               //step code                                             //do step
               ;
               IF #ContEnable = true THEN                               //enable continue function
                   #cont_enable[1] := true;
               END_IF;
               IF #EndOfStep = true THEN                                //define end of step condition
                   #end_of_step[1] := true;                            
               END_IF;                                    
               #next_step[1] := 0;                                      //define next step #
               IF #end_of_step[1] = true THEN                           //do on transition
                   //transition code
                   ;
               END_IF;

   //-step-100---level--1----------------------------------------------name-(remarks)----------------------                                                 
           100 :                                                     
               IF #next_step[1] = #active_step[1] THEN                   //init step     
                   //init code 
                   ;                                                  
               END_IF;

               //step code                                             //do step
               ;
               IF #ContEnable = true THEN                               //enable continue function
                   #cont_enable[1] := true;
               END_IF;
               IF #EndOfStep = true THEN                                //define end of step condition
                   #end_of_step[1] := true;                            
               END_IF;                                    
               #next_step[1] := 0;                                      //define next step #
               IF #end_of_step[1] = true THEN                           //do on transition
                   //transition code
                   ;
               END_IF;

   //-step-200---level--1----------------------------------------------name-(remarks)----------------------                                                 
           200 :                                                     
               IF #next_step[1] = #active_step[1] THEN                   //init step     
                   //init code 
                   ;                                                  
               END_IF;

               //step code                                             //do step
               ;
               IF #ContEnable = true THEN                               //enable continue function
                   #cont_enable[1] := true;
               END_IF;
               IF #EndOfStep = true THEN                                //define end of step condition
                   #end_of_step[1] := true;                            
               END_IF;                                    
               #next_step[1] := 0;                                      //define next step #
               IF #end_of_step[1] = true THEN                           //do on transition
                   //transition code
                   ;
               END_IF;

   //-error------level--1---------------------------------------------------(error in level 1)-------------
       ELSE:                                                        
           //error code                                                //do error code
           ;        
   //------------------------------------------------------------------------------------------------------
       END_CASE;

       CASE #active_step[2] OF    //sequence level_2
   //step--0-----level--2-------------------------------------------------off--(sequence off)--------------
           0    :                                                  
                #next_step[2] := 0;

   //step--1-----level--2-------------------------------------------------hold-(test sequence)-------------
           1   :                                                       
               IF #next_step[2] = #active_step[2] THEN                   //init step     
                   //init code
                   ; 
               END_IF;

               //step code                                             //do step
               ;

   //-step-10----level--2----------------------------------------------main-(start sequence)---------------                                                 
           10  :                                                     
               IF #next_step[2] = #active_step[2] THEN                   //init step     
                   //init code 
                   ;                                                  
               END_IF;

               //step code                                             //do step
               ;
               IF #ContEnable = true THEN                               //enable continue function
                   #cont_enable[2] := true;
               END_IF;
               IF #EndOfStep = true THEN                                //define end of step condition
                   #end_of_step[2] := true;                            
               END_IF;                                    
               #next_step[1] := 0;                                      //define next step #
               IF #end_of_step[2] = true THEN                           //do on transition
                   //transition code
                   ;
               END_IF;

   //-step-100---level--2----------------------------------------------name-(remarks)----------------------                                                 
           100 :                                                     
               IF #next_step[2] = #active_step[2] THEN                   //init step     
                   //init code 
                   ;                                                  
               END_IF;

               //step code                                             //do step
               ;
               IF #ContEnable = true THEN                               //enable continue function
                   #cont_enable[2] := true;
               END_IF;
               IF #EndOfStep = true THEN                                //define end of step condition
                   #end_of_step[2] := true;                            
               END_IF;                                    
               #next_step[2] := 0;                                      //define next step #
               IF #end_of_step[2] = true THEN                           //do on transition
                   //transition code
                   ;
               END_IF;

   //-error------level--2---------------------------------------------------(error in level 2)-------------
       ELSE:                                                        
           //error code                                                //do error code
           ;        
   //------------------------------------------------------------------------------------------------------
       END_CASE;

       //save crystal position at start of body - used in FB AM_RE
       //---------------------------------------------------------
       "AV".XT_POS_AT_START_BY   :=  #xt_pos_at_start;

       #start_previous := #start;                                    //save start input for next call 
       #cont_previous := "APC".CONT;                                  //save cont input for next call 
       #resume_previous := "APC".RESUME;                              //save resume input for next call
       #jump_previous := "APC".JUMP;                                  //save jump input for next call
       #single_previous := "APC".SINGLE;                              //save single input for next call
END_FUNCTION_BLOCK

FUNCTION_BLOCK "AM_EC"   // FB202, SCL
{ S7_Optimized_Access := 'FALSE' }
VERSION : 0.0
// --------------------------------------------------------------------------------
//     program     :    AM_EC
//     description :    apc endcone module  
//     name        :    D. Bruess
//     date        :    01.12.99
//     
//     revision    :    change default rotation direction: xtal= ccw and cruc= cw
//     name        :    G. Eibelsh鋟ser
//     date        :    26.04.00
// 
//     revision    :    
//     name        :    
//     date        :    
//                     (c)CGS
//     --------------------------------------------------------------------------------
   VAR_INPUT
      start : Bool;   // start sequence, activate step 10 (impulse triggered)
   END_VAR
   VAR
      start_previous : Bool;   // start input value of last call
      cont_previous : Bool;   // cont input value of last call
      resume_previous : Bool;   // resume input value of last call
      jump_previous : Bool;   // jump input value of last call
      single_previous : Bool;   // single input value of last call
      active_step : Array[0..7] of Int;   // active step number for sequence level 0..7
      next_step : Array[0..7] of Int;   // next step number for sequence level 0..7
      hold_step : Array[0..7] of Int;   // step number of step on hold
      end_of_step : Array[0..7] of Bool;   // active step is done flag for sequence 0..7
      EndOfStep : Bool;   // default value for active step is done flag
      cont_enable : Array[0..7] of Bool;   // enable continue function
      ContEnable : Bool;   // default value for enable continue function
      xt_pos_at_start : Real;   // crystal position at start of neck
      old_inc_xt_spd : Real;   // old increment value
      old_inc_cr_spd : Real;   // old increment value
      old_inc_xt_rot : Real;   // old increment value
      old_inc_cr_rot : Real;   // old increment value
   END_VAR
BEGIN


       "APC".STATUS := "APC".ENDCONE;                                  // set apc status               

       "AM_SEQUENCE_CTL" (start_p            := #start,               // control sequence
                        start_previous_p   := #start_previous,
                        cont_previous_p    := #cont_previous, 
                        resume_previous_p  := #resume_previous,
                        jump_previous_p    := #jump_previous,
                        single_previous_p  := #single_previous,
                        active_step_p      := #active_step, 
                        next_step_p        := #next_step,
                        hold_step_p        := #hold_step, 
                        end_of_step_p      := #end_of_step, 
                        cont_enable_p      := #cont_enable); 

       //Set the "Oxidation valve" in all Phases
       "DC".V21_OP:= DINT_TO_BOOL(REAL_TO_DINT("PAR_MAIN".EC_V21_OPEN));

       CASE #active_step[0] OF    //sequence level_0
   //step--0-----level--0-------------------------------------------------off--(sequence off)--------------
           0    :                                                  
                #next_step[0] := 0;

   //step--1-----level--0-------------------------------------------------hold-(test sequence)-------------
           1   :                                                       
               IF #next_step[0] = #active_step[0] THEN                   //init step     
                   //init code
                   ; 
               END_IF;

               //step code                                             //do step
               ;

   //-step-10----level--0----------------------------------------------main-(start sequence)---------------                                                 

   //-step-10----level--0-------------------------------------------------------------                                                 
   //            EC: init endcone sequence
   //---------------------------------------------------------------------------------                                                 
           10  :                                                  
               // save data of grown body (for 2nd body)
               // --------------------------------------
               IF ("APC".PNBDY = TRUE) THEN
                   "APC".LEN2_CALC := FALSE;
                   "CM_SAVE_GROWN_BY" (with_endcone := TRUE,
                                     dia          := "AC".SET_XT_DIA,
                                     len          := "AV".ACT_XT_LEN);
               END_IF;

               // init vacuum system
               // ------------------
               "DC".V1_OP    := TRUE;                         // open V1
               "DC".V3_OP    := FALSE;
               "DC".V4_OP    := FALSE;
               "DC".V5_OP    := TRUE;                         // open V5
               "DC".V6_OP    := FALSE;
               "DC".V8_OP    := FALSE;
               "DC".V11_OP   := FALSE;
               "DC".V11_CL   := TRUE;
               "DC".V12_OP   := FALSE;
               "DC".V13_OP   := FALSE;
               "DC".V20_OP   := FALSE;
               "DC".V22_OP   := FALSE;
               "DC".V24_OP   := FALSE;
               "DC".P1_ON    := TRUE;                         // start main pump
               "DC".P3_ON    := FALSE;
               "DC".V3_4_OP  := FALSE;
               "DC".V1_1_REL := FALSE;

               "DC".V1_OPEN_REQ   := FALSE;                // only EKZ 2700
               "DC".V1_CLOSE_REQ  := FALSE;

               "DC".V3_2_OP := FALSE;                      // vacuum valve feeder

               // init drives
               // -----------
               IF (("CNF".ACT_DVC_CNF AND 2#0100_0000_0000_0000_0000_0000_0000_0000) = 2#0100_0000_0000_0000_0000_0000_0000_0000) THEN   //gap control activated
                   ;                                   //direction is set in step 250 (related to gap control)
               ELSE
                   "DC".XT_LFT_UP := TRUE;               // crystal lift up - direction is set in step 250 (related to gap control)
                   "DC".XT_LFT_DN := FALSE;
                   "DC".CR_LFT_UP := TRUE;               // crucible lift up - direction is set in step 250 (related to gap control)
                   "DC".CR_LFT_DN := FALSE;
               END_IF;

               "DC".XT_LFT_FST := FALSE;
               "DC".XT_ROT_CW := "BM_ROT_DRV_DIR_DB".ROT_DIR;            //1 = cw
               "DC".XT_ROT_CCW := NOT "BM_ROT_DRV_DIR_DB".ROT_DIR;       //0 = ccw

               "DC".CR_LFT_FST := FALSE;
               "DC".CR_ROT_CW := NOT "BM_ROT_DRV_DIR_DB".ROT_DIR;        //0 = cw
               "DC".CR_ROT_CCW := "BM_ROT_DRV_DIR_DB".ROT_DIR;           //1 = ccw


               "AC".SET_XT_SPD := "CTL".SET_XT_SPD;                
               "AC".SET_XT_ROT := "KYA".SET_XT_ROT;
               "AC".SET_CR_SPD := "CTL".SET_CR_SPD;
               "AC".SET_CR_ROT := "KYA".SET_CR_ROT;

               // init heater
               // -----------
               "DC".HTR_1_ON := TRUE;                     // heater on
               "DC".HTR_2_ON := TRUE;
               "DC".HTR_3_ON := FALSE;

               // AC.SET_HTR_1_PWR := 0.0;                 do not set, loop is on
               // AC.SET_HTR_2_PWR := 0.0;
               // AC.SET_HTR_3_PWR := 0.0;

               //mobile feeder
               //-------------
               "DC".MOB_FDR_MVE_IN_SEQ_ON    :=  FALSE;
               IF ("LT".MOB_FDR_DCK_DONE AND ("DV".FDG_MVE_IN_SEQ_DONE OR NOT "DV".FDG_MVE_OUT_SEQ_DONE)) THEN 
                   "DC".MOB_FDR_MVE_OUT_SEQ_ON   :=  TRUE;
               ELSE
                   "DC".MOB_FDR_MVE_OUT_SEQ_ON   :=  FALSE;
               END_IF;
               "DC".MOB_FDR_VIB_ON           :=  FALSE;
               "FLT".MOB_FDR_NOT_DCK         :=  FALSE;
               "FLT".MOB_FDR_STP_PARA        :=  FALSE;

               // init magnet
               // -----------
               "DC".MAG_ON := ("AC".SET_MAG_1_CUR > 0.0);

               "AC".SET_MAG_1_CUR := "KYA".SET_MAG_1_CUR;
               "AC".SET_MAG_2_CUR := "KYA".SET_MAG_1_CUR * "KYA".SET_MAG_RATIO_CUR;

               // init control loops
               // ------------------
               "DC".CTL_DIA_ON       := FALSE;             // all control loops off
               "DC".CTL_GRW_RTE_ON   := FALSE;
               "DC".CTL_PULL_RTE_ON  := FALSE;
               "DC".CTL_CRUC_ROT_ON  := FALSE;
               "DC".CTL_MLT_LVL_ON   := FALSE;
               "DC".CTL_MLT_1_TMP_ON := FALSE;
               "DC".CTL_MLT_2_TMP_ON := FALSE;
               "DC".CTL_MLT_DRIFT_ON := FALSE;
               "DC".CTL_GAP_ON       := FALSE;

               "DC".CTL_HTR_1_TMP_ON := TRUE;              // heater temp loop on
               //  DC.CTL_HTR_2_TMP_ON := TRUE;

               "DC".SET_HTR_1_TMP_ABS := FALSE;                // enable inc functions
               "DC".SET_HTR_2_PWR_ABS := FALSE;


               "DC".CTL_PRS_ON := TRUE;                    // pressure control on

               "DC".CTL_SI_FDR_ON := FALSE;
               "DC".CTL_DOP_FDR_ON := FALSE;

               "DV".TRANS_SH_BY_FLAG := FALSE;
               "DV".START_SH_FLAG    := FALSE;

               "AC".SET_XT_DIA := 0.0;
               "AC".SET_GRW_RTE := 0.0;
               "AC".SET_AVG_SPD := 0.0;
               "AC".SET_AVG_CRUC_ROT := 0.0;
               "AC".SET_MLT_LVL_LSR := 0.0;
               "AC".SET_MLT_1_TMP := 0.0;
               "AC".SET_MLT_2_TMP := 0.0;

               // init measurement system
               // -----------------------
               "DC".CAM_ISP_ON   :=  TRUE;      //inspection on
               "DC".CAM_INIT     :=  FALSE;
               "DC".CAM_MLT      :=  TRUE;
               "DC".CAM_DIP      :=  FALSE;
               "DC".CAM_DIA      :=  FALSE;
               "DC".CAM_SEL_1    :=  TRUE;
               "DC".CAM_SEL_2    :=  FALSE;

               //set measurement window in upper left corner of image - no measurement required
               //------------------------------------------------------------------------------
               "AC".SET_SEN_THR    := 50.0;  
               "AC".SET_SEN_WDH    :=  5.0;        
               "AC".SET_SEN_HGT    :=  5.0;       
               "AC".SET_SEN_CTR_X  := 10.0;       
               "AC".SET_SEN_CTR_Y  := 10.0;  

               "DV".THR_CALC_DISABLED  := TRUE;      //threshold calculation in this step is disabled

               "DC".LSR_ON := FALSE;                       // laser off
               "DC".MCC_ON := FALSE;                       // melt contact control off
               "DC".MCC_TST_ON := FALSE;

               // init Si feeder system
               // ---------------------
               "DC".SI_FDR_ON := FALSE;                    // feeder off
               "DC".DOP_FDR_ON := FALSE;

               "AC".SET_FDR_SI := 0.0;
               "AC".SET_FDR_DOP := 0.0;

               // init lamp on control cabinet
               // ----------------------------
               "DV".LMP_OR := false;

               // save start position, reset length
               // ---------------------------------
               #xt_pos_at_start := "AV".ACT_XT_POS;
               "AV".ACT_XT_LEN_PRC := 0.0; 
               "AV".ACT_XT_LEN := 0.0;

               // calculate all setpoints 
               // -----------------------
               "AM_PAR_FNC_EC" (act_x_value := 0);



               // enable automatic mode
               // ---------------------
               "DC".MOD_AUT_ENB := TRUE;

               #end_of_step[0]  := true;                            
               #next_step[0]    := 100;

   //-step-100---level--0-------------------------------------------------------------                                                 
   //            EC: wait for automatic mode
   //---------------------------------------------------------------------------------                                                 
           100 :                                                     
               IF #next_step[0] = #active_step[0] THEN
                   "APC".OP_MSG := "OP_MSG".WAIT_FOR_AUTO;                                                  
               END_IF;

               // do not count the length while waiting for automatic
               // ---------------------------------------------------
               #xt_pos_at_start := "AV".ACT_XT_POS;
               "AV".ACT_XT_LEN_PRC := 0.0; 
               "AV".ACT_XT_LEN := 0.0;

               // calculate all setpoints 
               // -----------------------
               "AM_PAR_FNC_EC" (act_x_value := 0.0);

               IF "APC".AUTOMATIC = TRUE THEN                     // automatic mode ?
                   #end_of_step[0] := true;                            
               END_IF;                                    
               #next_step[0] := 200;

   //-step-200---level--0-------------------------------------------------------------                                                 
   //            EC: start time
   //---------------------------------------------------------------------------------                                                 
           200 :                                                     
               "APC".ACT_TME_PROC := 0;                           // start process time
               "APC".ACT_TME_STE := 0;                            // reset time of step
               "APC".TI[0] := 0;                                  // start waiting time
               "APC".OP_MSG := "OP_MSG".BLANK;                                                  

               #end_of_step[0] := true;

               IF (("CNF".ACT_DVC_CNF AND 2#0100_0000_0000_0000_0000_0000_0000_0000) = 2#0100_0000_0000_0000_0000_0000_0000_0000) THEN   //gap control activated
                   #next_step[0] := 250;
               ELSE
                   #next_step[0] := 300;
               END_IF;

   //-step-250---level--0-------------------------------------------------------------                                                 
   //            EC: set lifting direction related to speed set points
   //---------------------------------------------------------------------------------                                                 
           250 :                                                     
               //Set direction of crystal lift
               //-----------------------------
               IF (("CTL".SET_XT_SPD + "AV".MLT_LVL_SFT_OFFS_SPD + "CTL".SET_SPEED_OFFS) < 0.0) THEN
                   "DC".XT_LFT_UP    := FALSE;
                   "DC".XT_LFT_DN    := TRUE; // crystal lift down
                   "LT".XT_LFT_UP    := FALSE;
               ELSE
                   "DC".XT_LFT_UP    := TRUE; // crystal lift up
                   "DC".XT_LFT_DN    := FALSE;
                   "LT".XT_LFT_DN    := FALSE;
               END_IF;
               //Set direction of crucible lift
               //------------------------------
               IF (("CTL".SET_CR_SPD + "AV".MLT_LVL_SFT_OFFS_SPD + "CTL".SET_SPEED_OFFS ) < 0.0) THEN
                   "DC".CR_LFT_UP    := FALSE;
                   "DC".CR_LFT_DN    := TRUE; // Crucible lift down
                   "LT".CR_LFT_UP    := FALSE;
               ELSE
                   "DC".CR_LFT_UP    := TRUE; // Crucible lift up
                   "DC".CR_LFT_DN    := FALSE;
                   "LT".CR_LFT_DN    := FALSE;
               END_IF;

               //lifitng direction upwads active?
               // -------------------------------
               IF ("DC".XT_LFT_UP AND "DC".CR_LFT_UP) THEN    
                   #end_of_step[0] := true;                            
               END_IF;

               #next_step[0] := 300; 

   //-step-300---level--0-------------------------------------------------------------                                                 
   //            EC: do initial inc. for speed, rotation and heater
   //---------------------------------------------------------------------------------                                                 
           300 :                                                     
               IF #next_step[0] = #active_step[0] THEN                       
                   //display initial temperature and power setpoints
                   //-----------------------------------------------
                   "DIS".HTR_1_TMP_SET_PHA_STR   :=  "CTL".SET_HTR_1_TMP;
                   "DIS".HTR_2_PWR_SET_PHA_STR   :=  "CTL".SET_HTR_2_PWR;
                   // do heater inc.
                   // --------------
                   "DC".RSTRT_HTR_1_TMP_INC := TRUE;
                   "DC".RSTRT_HTR_2_PWR_INC := TRUE;
                   "AC".SET_HTR_1_TMP_INC := "AV".SET_HTR_1_TMP_INC;
                   "AC".SET_HTR_2_PWR_INC := "AV".SET_HTR_2_PWR_INC;
               END_IF;

               // calculate actual length
               // -----------------------
               "AM_CALC_LENGTH" (start_pos := #xt_pos_at_start,
                               actual_pos := "AV".ACT_XT_POS,
                               total_len := "PAR_MAIN".EC_XT_LEN,
                               actual_len => "AV".ACT_XT_LEN,
                               actual_len_prc => "AV".ACT_XT_LEN_PRC);


               // calculate all setpoints for this step
               // -------------------------------------                                      
               "AM_PAR_FNC_EC" (act_x_value := "AV".ACT_XT_LEN);

               // setpoint magnet
               // ---------------
               "DC".MAG_ON := ("AC".SET_MAG_1_CUR > 0.0);

               "AC".SET_MAG_1_CUR := "AV".SET_MAG_1_CUR;
               "AC".SET_MAG_2_CUR := "AV".SET_MAG_1_CUR * "AV".SET_MAG_RATIO_CUR;



               // reset waiting time 1 for oxidation process
               //-------------------------------------------
               "APC".TI[1] := 0;

               // wait ?
               // ------
               IF ("APC".TI[0] > 3) THEN    
                   #end_of_step[0] := true;                            
               END_IF;
               #next_step[0] := 400; 


   //-step-400---level--0-------------------------------------------------------------                                                 
   //            EC: do endcone process
   //---------------------------------------------------------------------------------                                                 
           400 :                                                  
               IF #next_step[0] = #active_step[0] THEN                       
                   // init inc. functions
                   // -------------------
                   #old_inc_xt_spd := 0.0;
                   #old_inc_cr_spd := 0.0;
                   #old_inc_xt_rot := 0.0;
                   #old_inc_cr_rot := 0.0;
               END_IF;

               // calculate actual length
               // -----------------------
               "AM_CALC_LENGTH" (start_pos      := #xt_pos_at_start,
                               actual_pos     := "AV".ACT_XT_POS,
                               total_len      := "PAR_MAIN".EC_XT_LEN,
                               actual_len     => "AV".ACT_XT_LEN,
                               actual_len_prc => "AV".ACT_XT_LEN_PRC);

               // calculate all setpoints for this step
               // -------------------------------------                                      
               "AM_PAR_FNC_EC" (act_x_value := "AV".ACT_XT_LEN);

               // setpoint magnet
               // ---------------
               "DC".MAG_ON := ("AC".SET_MAG_1_CUR > 0.0);

               "AC".SET_MAG_1_CUR := "AV".SET_MAG_1_CUR;
               "AC".SET_MAG_2_CUR := "AV".SET_MAG_1_CUR * "AV".SET_MAG_RATIO_CUR;

               // increment function for speed and rotation
               // -----------------------------------------
               "AM_CALC_INC" (inc_disable := FALSE,
                            semi        := "SY".CTL_DIA_SMI,     // semi mode for crystal lift
                            inc_new     := "AV".SET_XT_SPD,
                            setp_man    := "KYA".SET_XT_SPD,
                            setp_min    := 0.0,                
                            setp_max    := "CNF".XT_LFT_RANGE,
                            setp_out    := "AC".SET_XT_SPD,
                            inc_old     := #old_inc_xt_spd );

               "AM_CALC_INC" (inc_disable := FALSE,
                            semi        := "SY".CTL_CR_SPD_SMI,
                            inc_new     := "AV".SET_CR_SPD,
                            setp_man    := "KYA".SET_CR_SPD,
                            setp_min    := 0.0,
                            setp_max    := "CNF".CR_LFT_RANGE,
                            setp_out    := "AC".SET_CR_SPD,
                            inc_old     := #old_inc_cr_spd );

               "AM_CALC_INC" (inc_disable := ("PAR_MAIN".EC_ROT_ABS_INC = 1.0), 
                            semi        := "SY".CTL_XT_ROT_SMI,  
                            inc_new     := "AV".SET_XT_ROT,
                            setp_man    := "KYA".SET_XT_ROT,
                            setp_min    := 0.0,
                            setp_max    := "CNF".XT_ROT_RANGE,
                            setp_out    := "AC".SET_XT_ROT,
                            inc_old     := #old_inc_xt_rot );

               "AM_CALC_INC" (inc_disable := ("PAR_MAIN".EC_ROT_ABS_INC = 1.0),
                            semi        := "SY".CTL_CR_ROT_SMI,  
                            inc_new     := "AV".SET_CR_ROT,
                            setp_man    := "KYA".SET_CR_ROT,
                            setp_min    := 0.0,
                            setp_max    := "CNF".CR_ROT_RANGE,
                            setp_out    := "AC".SET_CR_ROT,
                            inc_old     := #old_inc_cr_rot );

               // heater temp/power inc.
               // ----------------------
               "AC".SET_HTR_1_TMP_INC := "AV".SET_HTR_1_TMP_INC;
               "AC".SET_HTR_2_PWR_INC := "AV".SET_HTR_2_PWR_INC;

               // melt contact control
               // --------------------   
               "DC".MCC_ON := ("PAR_MAIN".EC_MLT_CONTACT_CTL = 1.0);     

               // endcone length reached ?
               // ------------------------
               IF ("AV".ACT_XT_LEN >= "PAR_MAIN".EC_XT_LEN) THEN    
                   #end_of_step[0] := true;                            
               END_IF;
               #next_step[0] := 500;


   //-step-500---level--0-------------------------------------------------------------                                                 
   //            EC: start shut down process
   //---------------------------------------------------------------------------------                                                 
           500 :                                                  
               IF #next_step[0] = #active_step[0] THEN
                   "APC".OP_MSG := "OP_MSG".BLANK;
               END_IF;

               IF ("APC".SUTDN = TRUE) THEN
                   "DC".MOD_SD := TRUE;                           // switch to shut down 
               ELSE
                   "DC".MOD_RE := TRUE;                           // switch to removal 
               END_IF;   
               #next_step[0] := 500;                             // E N D 



   //---------------------------------------------------------------------------------                                                 
   //-error------level--0---------------------------------------------------(error in level 0)-------------
       ELSE:                                                        
           //error code                                                //do error code
           ;        
   //------------------------------------------------------------------------------------------------------
       END_CASE;

       #start_previous := #start;                                    //save start input for next call 
       #cont_previous := "APC".CONT;                                  //save cont input for next call 
       #resume_previous := "APC".RESUME;                              //save resume input for next call
       #jump_previous := "APC".JUMP;                                  //save jump input for next call
       #single_previous := "APC".SINGLE;                              //save single input for next call
END_FUNCTION_BLOCK

FUNCTION_BLOCK "AM_SD"   // FB203, SCL
{ S7_Optimized_Access := 'FALSE' }
VERSION : 0.0
// --------------------------------------------------------------------------------
//     program     :    AM_SD
//     description :    apc shut down module  
//     name        :    D. Bruess
//     date        :    18.11.99
//     
//     revision    :    change default rotation direction: xtal= ccw and cruc= cw
//     name        :    G. Eibelsh鋟ser
//     date        :    26.04.00
// 
//     revision    :    
//     name        :    
//     date        :    
//                     (c)PVA TePla AG
//     --------------------------------------------------------------------------------
   VAR_INPUT
      start : Bool;   // start sequence, activate step 10 (impulse triggered)
   END_VAR
   VAR
      start_previous : Bool;   // start input value of last call
      cont_previous : Bool;   // cont input value of last call
      resume_previous : Bool;   // resume input value of last call
      jump_previous : Bool;   // jump input value of last call
      single_previous : Bool;   // single input value of last call
      active_step : Array[0..7] of Int;   // active step number for sequence level 0..7
      next_step : Array[0..7] of Int;   // next step number for sequence level 0..7
      hold_step : Array[0..7] of Int;   // step number of step on hold
      end_of_step : Array[0..7] of Bool;   // active step is done flag for sequence 0..7
      EndOfStep : Bool;   // default value for active step is done flag
      cont_enable : Array[0..7] of Bool;   // enable continue function
      ContEnable : Bool;   // default value for enable continue function
      cruc_in_pos : Bool;   // crucible in new position
      xtal_in_pos : Bool;   // crystal in new position
      prs_ctl_done : Bool;   // new pressure reached
      v4_lim_reached : Bool;   // pressure limit for gas inlet through V4 is reached
      OV2 : Bool;   // ???????
      par_line : Int;   // act. line from parameter table
      par_step : Int;   // number of this step
      par_time : Int;   // time parameter for this step
      set_cr_pos_old : Real;   // old setpoint for crucible position
      set_xt_pos_old : Real;   // old setpoint for crystal position
      set_clf_prs_old : Real;   // old setpoint for pressure
      set_gas_1_flw_old : Real;   // old setpoint for gas flow
      set_gas_2_flw_old : Real;   // old setpoint for gas flow
      prs_leak_test_start : Real;   // pressure at start of leak test
   END_VAR
BEGIN


       "APC".STATUS := "APC".SHUT_DOWN;                                // set apc status               

       "AM_SEQUENCE_CTL" (start_p            := #start,               // control sequence
                        start_previous_p   := #start_previous,
                        cont_previous_p    := #cont_previous, 
                        resume_previous_p  := #resume_previous,
                        jump_previous_p    := #jump_previous,
                        single_previous_p  := #single_previous,
                        active_step_p      := #active_step, 
                        next_step_p        := #next_step,
                        hold_step_p        := #hold_step, 
                        end_of_step_p      := #end_of_step, 
                        cont_enable_p      := #cont_enable); 


       CASE #active_step[0] OF    //sequence level_0
   //step--0-----level--0-------------------------------------------------off--(sequence off)--------------
           0    :                                                  
                #next_step[0] := 0;

   //step--1-----level--0-------------------------------------------------hold-(test sequence)-------------
           1   :                                                       
               IF #next_step[0] = #active_step[0] THEN                   //init step     
                   //init code
                   ; 
               END_IF;

               //step code                                             //do step
               ;

   //-step-10----level--0----------------------------------------------main-(start sequence)---------------                                                 

   //-step-10----level--0-------------------------------------------------------------                                                 
   //            SD: init shut down sequence
   //---------------------------------------------------------------------------------                                                 
           10  :                                                     

               // init vacuum system
               // ------------------
               "DC".V3_OP    := FALSE;
               "DC".V3_2_OP  := FALSE;                      // vacuum valve feeder
               "DC".V4_OP    := FALSE;
               "DC".V5_OP    := TRUE;                         // open V5
               "DC".V6_OP    := FALSE;
               "DC".V8_OP    := FALSE;
               "DC".V11_OP   := FALSE;
               "DC".V11_CL   := TRUE;
               "DC".V12_OP   := FALSE;
               "DC".V13_OP   := FALSE;
               "DC".V20_OP   := FALSE;
               "DC".V21_OP   := DINT_TO_BOOL(REAL_TO_DINT("PAR_MAIN".SD_V21_OPEN));    //Set the Oxidation valve according parameter
               "DC".V22_OP   := FALSE;
               "DC".V24_OP   := FALSE;
               "DC".P1_ON    := TRUE;                         // start main pump
               "DC".P3_ON    := FALSE;
               "DC".V1_OPEN_REQ   := FALSE;                // only EKZ 2700
               "DC".V1_CLOSE_REQ  := FALSE;
               "DC".V3_4_OP  := FALSE;
               "DC".V1_1_REL := FALSE;

               #set_clf_prs_old  := -1.0; 
               #set_gas_1_flw_old:= -1.0;
               #set_gas_2_flw_old:= -1.0;
               #prs_ctl_done := FALSE;
               "AM_PRS_CTRL_DB".req_vac := FALSE;
               "AM_PRS_CTRL_DB".req_vent := FALSE;

               // init drives
               // -----------
               "DC".XT_LFT_UP  := FALSE;                    // stop crystal lift
               "DC".XT_LFT_DN  := FALSE;
               "DC".XT_LFT_FST := FALSE;
               "DC".XT_ROT_CW  := "BM_ROT_DRV_DIR_DB".ROT_DIR      AND ("AC".SET_XT_ROT <> 0.0);    //1 = cw
               "DC".XT_ROT_CCW := NOT "BM_ROT_DRV_DIR_DB".ROT_DIR  AND ("AC".SET_XT_ROT <> 0.0);    //0 = ccw


               "DC".CR_LFT_UP  := FALSE;                    // stop crucible lift
               "DC".CR_LFT_DN  := FALSE;
               "DC".CR_LFT_FST := FALSE;
               "DC".CR_ROT_CW  := NOT "BM_ROT_DRV_DIR_DB".ROT_DIR  AND ("AC".SET_CR_ROT <> 0.0);     //0 = cw
               "DC".CR_ROT_CCW := "BM_ROT_DRV_DIR_DB".ROT_DIR      AND ("AC".SET_CR_ROT <> 0.0);     //1 = ccw


               "AC".SET_XT_SPD := 0.0;                
               "AC".SET_XT_ROT := "KYA".SET_XT_ROT;
               "AC".SET_CR_SPD := 0.0;
               "AC".SET_CR_ROT := "KYA".SET_CR_ROT;

               #set_cr_pos_old := -1.0;
               #set_xt_pos_old := -1.0;
               #cruc_in_pos := FALSE;
               #xtal_in_pos := FALSE;
               "AM_CR_DRV_MOVE_DB".pos_req := FALSE;
               "AM_XT_DRV_MOVE_DB".pos_req := FALSE;

               // init heater
               // -----------
               "DC".HTR_1_ON := ("AC".SET_HTR_1_PWR > 0.0);    // heater on
               "DC".HTR_2_ON := FALSE;                       // heater off
               "DC".HTR_3_ON := FALSE;

               "AC".SET_HTR_1_PWR := "KYA".SET_HTR_1_PWR;
               "AC".SET_HTR_2_PWR := 0.0;
               "AC".SET_HTR_3_PWR := 0.0;

               //mobile feeder
               //-------------
               "DC".MOB_FDR_MVE_IN_SEQ_ON    :=  FALSE;
               IF ("LT".MOB_FDR_DCK_DONE AND ("DV".FDG_MVE_IN_SEQ_DONE OR NOT "DV".FDG_MVE_OUT_SEQ_DONE)) THEN 
                   "DC".MOB_FDR_MVE_OUT_SEQ_ON   :=  TRUE;
               ELSE
                   "DC".MOB_FDR_MVE_OUT_SEQ_ON   :=  FALSE;
               END_IF;
               "DC".MOB_FDR_VIB_ON           :=  FALSE;
               "FLT".MOB_FDR_NOT_DCK         :=  FALSE;
               "FLT".MOB_FDR_STP_PARA        :=  FALSE;

               // init magnet
               // -----------
               "DC".MAG_ON := ("AC".SET_MAG_1_CUR > 0.0);

               "AC".SET_MAG_1_CUR := "KYA".SET_MAG_1_CUR;            
               "AC".SET_MAG_2_CUR := "KYA".SET_MAG_1_CUR * "KYA".SET_MAG_RATIO_CUR;

               // init control loops
               // ------------------
               "DC".CTL_DIA_ON := FALSE;                   // all control loops off
               "DC".CTL_GRW_RTE_ON := FALSE;
               "DC".CTL_PULL_RTE_ON := FALSE;
               "DC".CTL_CRUC_ROT_ON := FALSE;
               "DC".CTL_MLT_LVL_ON := FALSE;
               "DC".CTL_MLT_1_TMP_ON := FALSE;
               "DC".CTL_MLT_2_TMP_ON := FALSE;
               "DC".CTL_MLT_DRIFT_ON := FALSE;
               "DC".CTL_GAP_ON       := FALSE;

               "DC".CTL_HTR_1_TMP_ON := FALSE;
               // DC.CTL_HTR_2_TMP_ON := FALSE;

               "DC".SET_HTR_1_TMP_ABS := TRUE;             // disable inc functions
               "DC".SET_HTR_2_PWR_ABS := TRUE;


               "DC".CTL_PRS_ON := TRUE;                    // pressure control on

               "DC".CTL_SI_FDR_ON := FALSE;
               "DC".CTL_DOP_FDR_ON := FALSE;

               "DV".TRANS_SH_BY_FLAG := FALSE;
               "DV".START_SH_FLAG    := FALSE;


               "AC".SET_XT_DIA := 0.0;
               "AC".SET_GRW_RTE := 0.0;
               "AC".SET_AVG_SPD := 0.0;
               "AC".SET_AVG_CRUC_ROT := 0.0;
               "AC".SET_MLT_LVL_LSR := 0.0;
               "AC".SET_MLT_1_TMP := 0.0;
               "AC".SET_MLT_2_TMP := 0.0;
               "AC".SET_HTR_1_TMP := 0.0;
               "AC".SET_HTR_2_TMP := 0.0;

               // init measurement system
               // -----------------------
               "DC".CAM_ISP_ON   :=  FALSE;      //inspection off
               "DC".CAM_INIT     :=  FALSE;
               //DC.CAM_MLT      :=  FALSE;
               //DC.CAM_DIP      :=  FALSE;
               //DC.CAM_DIA      :=  TRUE;
               "DC".CAM_SEL_1    :=  TRUE;
               "DC".CAM_SEL_2    :=  FALSE;

               "DV".THR_CALC_DISABLED  := TRUE;      //threshold calculation in this step is disabled


               "DC".LSR_ON := FALSE;                       // laser off
               "DC".MCC_ON := FALSE;                       // melt contact control off
               "DC".MCC_TST_ON := FALSE;

               // init Si feeder system
               // ---------------------
               "DC".SI_FDR_ON := FALSE;                    // feeder off
               "DC".DOP_FDR_ON := FALSE;

               "AC".SET_FDR_SI := 0.0;
               "AC".SET_FDR_DOP := 0.0;

               // init lamp on control cabinet
               // ----------------------------
               "DV".LMP_OR := false;

               // calculate all setpoints (step no from 1st line of seqence table)
               // ----------------------------------------------------------------
               #par_line := 1;
               #par_step := REAL_TO_INT ("PAR_X_VALUES_1".PAR["APC".SHUT_DOWN, #par_line]);            
               "AM_PAR_FNC_SD" (act_x_value := #par_step);

               // process control flags
               // ---------------------
               "APC".PNBDY := FALSE;

               IF ("STA".ACT_STATE = "APC".STATE_RUN) THEN 
                   "DV".FIL_FSH_REQ_AFTER_SD :=  TRUE;           //request automtic filter flushing after shut down
               ELSE
                   "DV".FIL_FSH_REQ_AFTER_SD :=  FALSE;
               END_IF;

               // enable automatic mode
               // ---------------------
               "DC".MOD_AUT_ENB := TRUE;

               #end_of_step[0] := true;                            
               #next_step[0] := 100;


   //-step-100---level--0-------------------------------------------------------------                                                 
   //            SD: wait for automatic mode
   //---------------------------------------------------------------------------------                                                 
           100 :                                                     
               IF #next_step[0] = #active_step[0] THEN
                   "APC".OP_MSG := "OP_MSG".WAIT_FOR_AUTO;                                                  
               END_IF;

               IF "APC".AUTOMATIC = TRUE THEN                     // automatic mode ?
                   #end_of_step[0] := true;                            
               END_IF;                                    
               #next_step[0] := 150;


   //-step-150---level--0-------------------------------------------------------------                                                 
   //            SD: start time
   //---------------------------------------------------------------------------------                                                 
           150 :                                                     
               "APC".ACT_TME_PROC := 0;                           // start process time
               "APC".TI[1] := 0;                                  // reset waiting time 1 for oxidation process
               #end_of_step[0] := true;                            
               #next_step[0] := 200;


   //-step-200---level--0-------------------------------------------------------------                                                 
   //            SD: do one shut down step
   //---------------------------------------------------------------------------------                                                 
           200 :                                                     
               IF #next_step[0] = #active_step[0] THEN                       
                   //reset initial temperature and power setpoints
                   //---------------------------------------------
                   "DIS".HTR_1_TMP_SET_PHA_STR   :=  0.0;
                   "DIS".HTR_2_PWR_SET_PHA_STR   :=  0.0;

                   "APC".TI[0] := 0;                     // start step time
               END_IF;

               // fetch actual step number and time for this step
               // -----------------------------------------------
               #par_step := REAL_TO_INT ("PAR_X_VALUES_1".PAR["APC".SHUT_DOWN, #par_line]);            
               #par_time := REAL_TO_INT ("PAR_TME".PAR["APC".SHUT_DOWN, #par_line]);

               //Oxidation valve vacuum pipes
               //----------------------------
               "DC".V21_OP:= DINT_TO_BOOL(REAL_TO_DINT("PAR_MAIN".SD_V21_OPEN));

               // show actual step number
               // -----------------------
               "APC".OP_MSG := #par_step;

               // calculate all setpoints for this step
               // -------------------------------------                                      
               "AM_PAR_FNC_SD" (act_x_value := #par_step);

               // setpoint magnet
               // ---------------
               "DC".MAG_ON := ("AC".SET_MAG_1_CUR > 0.0);

               "AC".SET_MAG_1_CUR := "AV".SET_MAG_1_CUR;
               "AC".SET_MAG_2_CUR := "AV".SET_MAG_1_CUR * "AV".SET_MAG_RATIO_CUR;

               // move crucible
               // -------------
               IF ("AV".SET_CR_POS <> #set_cr_pos_old) THEN
                 #cruc_in_pos := FALSE;
               END_IF;

               "DC".CR_LFT_FST := TRUE;

               "AM_CR_DRV_MOVE_DB" ( set_pos := "AV".SET_CR_POS,
                                               set_spd := "AV".SET_CR_SPD,
                                               act_pos := "AV".ACT_CR_POS,
                                               cnf     := "CNF".CNF_CR_POS,
                                               out_up  := "DC".CR_LFT_UP,
                                               out_dn  := "DC".CR_LFT_DN,
                                               out_spd := "AC".SET_CR_SPD,
                                               done    := #cruc_in_pos);

               IF (#cruc_in_pos) THEN
                 #set_cr_pos_old := "AV".SET_CR_POS;
               END_IF;


               // move crystal
               // ------------
               IF ("AV".SET_XT_POS <> #set_xt_pos_old) THEN
                 #xtal_in_pos := FALSE;
               END_IF;

               "DC".XT_LFT_FST := TRUE;

               "AM_XT_DRV_MOVE_DB" (set_pos := "AV".SET_XT_POS,
                                           set_spd := - "AV".SET_XT_SPD,
                                           act_pos := "AV".ACT_XT_POS,
                                           cnf     := "CNF".CNF_XT_POS,
                                           out_up  := "DC".XT_LFT_DN,    // (!)
                                           out_dn  := "DC".XT_LFT_UP,    // (!)
                                           out_spd := "AC".SET_XT_SPD,
                                           done    := #xtal_in_pos);

               IF (#xtal_in_pos) THEN
                 #set_xt_pos_old := "AV".SET_XT_POS;
               END_IF;

               // control pressure and gas flow
               // -----------------------------
               IF ("AV".SET_GAS_1_FLW <> #set_gas_1_flw_old) THEN
                 #prs_ctl_done := FALSE;
               END_IF;
               IF ("AV".SET_GAS_2_FLW <> #set_gas_2_flw_old) THEN
                 #prs_ctl_done := FALSE;
               END_IF;
               IF ("AV".SET_PRS_FCH <> #set_clf_prs_old) THEN
                 #prs_ctl_done := FALSE;
               END_IF;

               "AM_PRS_CTRL_DB" (set_prs      := "AV".SET_PRS_FCH,
                                           set_flw_1    := "AV".SET_GAS_1_FLW,
                                           set_flw_2    := "AV".SET_GAS_2_FLW,
                                           act_prs      := "AV".ACT_PRS_FCH,
                                           out_V4       := "DC".V4_OP,
                                           out_V5       := "DC".V5_OP,
                                           out_prs_ctl  := "DC".CTL_PRS_ON,
                                           out_flw_1    := "AC".SET_GAS_1_FLW,
                                           out_flw_2    := "AC".SET_GAS_2_FLW,
                                           out_prs      := "AC".SET_CLF_PRS,
                                           out_valve_pos:= "AC".SET_CTL_VALVE_POS,
                                           done         := #prs_ctl_done);

               IF (#prs_ctl_done) THEN
                 #set_gas_1_flw_old := "AV".SET_GAS_1_FLW;
                 #set_gas_2_flw_old := "AV".SET_GAS_2_FLW;
                 #set_clf_prs_old := "AV".SET_PRS_FCH;
               END_IF;

               // close pressure control valve (only EKZ 2700)
               //---------------------------------------------
               IF "DC".CTL_PRS_ON = FALSE    THEN             
                   "DC".V1_OPEN_REQ   := FALSE;                
                   "DC".V1_CLOSE_REQ  := TRUE;
               ELSE
                   "DC".V1_OPEN_REQ   := FALSE;                
                   "DC".V1_CLOSE_REQ  := FALSE;
               END_IF;    

               // control heater
               // --------------
               "DC".HTR_1_ON := ("AC".SET_HTR_1_PWR > 0.0);
               "DC".HTR_2_ON := FALSE;


               // control rotation
               // ----------------
               "DC".XT_ROT_CW  := "BM_ROT_DRV_DIR_DB".ROT_DIR      AND ("AC".SET_XT_ROT <> 0.0);    //1 = cw
               "DC".XT_ROT_CCW := NOT "BM_ROT_DRV_DIR_DB".ROT_DIR  AND ("AC".SET_XT_ROT <> 0.0);    //0 = ccw
               "DC".CR_ROT_CW  := NOT "BM_ROT_DRV_DIR_DB".ROT_DIR  AND ("AC".SET_CR_ROT <> 0.0);    //0 = cw
               "DC".CR_ROT_CCW := "BM_ROT_DRV_DIR_DB".ROT_DIR      AND ("AC".SET_CR_ROT <> 0.0);    //1 = ccw


               // time till end of this step
               // --------------------------
               "APC".ACT_TME_STE := #par_time - "APC".TI[0];

               // end of step ?
               // -------------
               IF (("APC".TI[0] > #par_time)
                    AND (#cruc_in_pos = TRUE)
                    AND (#xtal_in_pos = TRUE)
                    AND (#prs_ctl_done = TRUE))  THEN

                  #end_of_step[0] := true;
               END_IF;

               #next_step[0] := 300; 


   //-step-300---level--0-------------------------------------------------------------                                                 
   //            SD: transition to next step, check for last step
   //---------------------------------------------------------------------------------                                                 
           300 :                                                  
               IF #next_step[0] = #active_step[0] THEN                       
                   // next line in parameter table
                   // ----------------------------
                   #par_line := #par_line + 1;
               END_IF;

               // fetch step number of this new line
               // ----------------------------------
               IF (#par_line <= 21) THEN
                   #par_step := REAL_TO_INT ("PAR_X_VALUES_1".PAR["APC".SHUT_DOWN, #par_line]);            
               END_IF;


               // step number = 0 or last line ? 
               // ------------------------------
               IF ((#par_step = 0)
                   OR (#par_line > 21) ) THEN

                   // start waiting time
                   // ------------------
                   #end_of_step[0] := true;                            
                   #next_step[0] := 400; 
               ELSE
                   // continue with next shut down step
                   // ---------------------------------
                   #end_of_step[0] := true;                            
                   #next_step[0] := 200; 
               END_IF;


   //-step-400---level--0-------------------------------------------------------------                                                 
   //            SD: initialisation after sequence
   //---------------------------------------------------------------------------------                                                 
           400 :                                                  
               IF #next_step[0] = #active_step[0] THEN
                   "APC".OP_MSG := "OP_MSG".PD_FINAL;
               END_IF;

               // set vacuum system
               // -----------------
               "DC".V3_OP    := FALSE;
               "DC".V3_2_OP  := FALSE;
               "DC".V4_OP    := FALSE;
               "DC".V5_OP    := FALSE;
               "DC".V6_OP    := FALSE;
               "DC".V8_OP    := FALSE;
               "DC".V11_OP   := FALSE;
               "DC".V11_CL   := FALSE;
               "DC".V12_OP   := FALSE;
               "DC".V13_OP   := FALSE;
               "DC".V24_OP   := FALSE;
               "DC".V21_OP   := FALSE;
               "DC".P1_ON    := TRUE;                         // pump on !!!   
               "DC".P3_ON    := FALSE;
               "DC".V1_OPEN_REQ   := FALSE;                // only EKZ 2700 old type
               "DC".V1_CLOSE_REQ  := TRUE;


               "AC".SET_CTL_VALVE_POS := 0.0;              // close throttle valve
               "AC".SET_GAS_1_FLW := 0.0;
               "AC".SET_GAS_2_FLW := 0.0;

               // stop drives
               // -----------
               "DC".XT_LFT_UP := FALSE;                    // stop crystal lift
               "DC".XT_LFT_DN := FALSE;
               "DC".XT_LFT_FST := FALSE;
               "DC".XT_ROT_CW := FALSE;                    // stop rotation
               "DC".XT_ROT_CCW := FALSE;

               "DC".CR_LFT_UP := FALSE;                    // stop crucible lift
               "DC".CR_LFT_DN := FALSE;
               "DC".CR_LFT_FST := FALSE;
               "DC".CR_ROT_CW := FALSE;                    // stop rotation
               "DC".CR_ROT_CCW := FALSE;

               "AC".SET_XT_SPD := 0.0;
               "AC".SET_XT_ROT := 0.0;
               "AC".SET_CR_SPD := 0.0;
               "AC".SET_CR_ROT := 0.0;

               // heater off
               // ----------
               "DC".HTR_1_ON := FALSE;                    // heater off
               "DC".HTR_2_ON := FALSE;
               "DC".HTR_3_ON := FALSE;

               "AC".SET_HTR_1_PWR := 0.0;
               "AC".SET_HTR_2_PWR := 0.0;
               "AC".SET_HTR_3_PWR := 0.0;

               // magnet off
               // ----------
               "DC".MAG_ON := FALSE;                       // magnet off

               "AC".SET_MAG_1_CUR := 0.0;
               "AC".SET_MAG_2_CUR := 0.0;

               // control loops off
               // -----------------
               "DC".CTL_DIA_ON := FALSE;                   // all control loops off
               "DC".CTL_GRW_RTE_ON := FALSE;
               "DC".CTL_PULL_RTE_ON := FALSE;
               "DC".CTL_MLT_LVL_ON := FALSE;
               "DC".CTL_MLT_1_TMP_ON := FALSE;
               "DC".CTL_MLT_2_TMP_ON := FALSE;

               "DC".CTL_HTR_1_TMP_ON := FALSE;
               "DC".CTL_HTR_2_TMP_ON := FALSE;

               "DC".CTL_PRS_ON := FALSE;                   // pressure control off

               "DC".CTL_SI_FDR_ON := FALSE;
               "DC".CTL_DOP_FDR_ON := FALSE;

               "AC".SET_XT_DIA := 0.0;
               "AC".SET_GRW_RTE := 0.0;
               "AC".SET_AVG_SPD := 0.0;
               "AC".SET_MLT_LVL_LSR := 0.0;
               "AC".SET_MLT_1_TMP := 0.0;
               "AC".SET_MLT_2_TMP := 0.0;
               "AC".SET_HTR_1_TMP := 0.0;
               "AC".SET_HTR_2_TMP := 0.0;

               // measurement system
               // ------------------
               "DC".CAM_ISP_ON   :=  FALSE;      //inspection off
               "DC".CAM_INIT     :=  FALSE;
               "DC".CAM_MLT      :=  FALSE;
               "DC".CAM_DIP      :=  FALSE;
               "DC".CAM_DIA      :=  TRUE;
               "DC".CAM_SEL_1    :=  TRUE;
               "DC".CAM_SEL_2    :=  FALSE;

               "DC".LSR_ON := FALSE;                       // laser off
               "DC".MCC_ON := FALSE;                       // melt contact control off
               "DC".MCC_TST_ON := FALSE;

               // init Si feeder system
               // ---------------------
               "DC".SI_FDR_ON := FALSE;                    // feeder off
               "DC".DOP_FDR_ON := FALSE;

               "AC".SET_FDR_SI := 0.0;
               "AC".SET_FDR_DOP := 0.0;


               // start waiting time
               // ------------------
               "APC".TI[0] := 0;

               #end_of_step[0] := TRUE;                            
               #next_step[0] := 500; 


   //-step-500---level--0-------------------------------------------------------------                                                 
   //            SD: waiting time after sequence
   //---------------------------------------------------------------------------------                                                 
           500 :                                                  
               // time till end of this step
               // --------------------------
               #par_time := REAL_TO_INT ("PAR_MAIN".SD_TME_TILL_VENT);
               "APC".ACT_TME_STE := #par_time - "APC".TI[0];

               // wait time reached ?
               // -------------------
               IF ("APC".TI[0] >= #par_time) THEN 
                   #end_of_step[0] := TRUE;                            
               END_IF;

               // set V2.1, V2.2
               // --------------
               "AM_SET_V2"(act_phase := "APC".SHUT_DOWN);

               IF ("PAR_MAIN".SD_LEAKTEST_TME = 0.0) THEN
                   // no leak test, switch to idle
                   // ----------------------------
                   "APC".OP_MSG := "OP_MSG".SD_WAIT_TILL_VENTING;
                   #next_step[0] := 950; 
               ELSE
                  // with leak test
                  // -------------- 
                  "APC".OP_MSG := "OP_MSG".SD_WAIT_TILL_LEAK_TEST;
                   #next_step[0] := 600; 
               END_IF;

   //-step-600---level--0-------------------------------------------------------------                                                 
   //            SD: pump down to final pressure
   //---------------------------------------------------------------------------------                                                 
           600 :                                                  
               IF #next_step[0] = #active_step[0] THEN
                   "APC".OP_MSG := "OP_MSG".PD_FINAL;
                   "DC".P1_ON := TRUE;                            // start main pump
                   "AC".SET_CTL_VALVE_POS := 100.0;               // open throttle valve
                   "DC".V1_OPEN_REQ   := TRUE;                    // only EKZ 2700
                   "DC".V1_CLOSE_REQ  := FALSE;

               END_IF;

               // set V2.1, V2.2
               // --------------
               "AM_SET_V2"(act_phase := "APC".SHUT_DOWN);


               IF ("AV".ACT_PRS_FCH < "PAR_MAIN".SD_FINAL_PRS) THEN     // final presssure ? 
                   #end_of_step[0] := true;                            
               END_IF;

               #next_step[0] := 700; 


   //-step-700---level--0-------------------------------------------------------------                                                 
   //            SD: close vacuum valve
   //---------------------------------------------------------------------------------                                                 
           700 :                                                  
               IF #next_step[0] = #active_step[0] THEN                       
                   "APC".OP_MSG := "OP_MSG".PD_LEAK_TEST;
               END_IF;

               "AC".SET_CTL_VALVE_POS := 0.0;                     // close throttle valve
               "DC".V1_OPEN_REQ   := FALSE;                       // only EKZ 2700
               "DC".V1_CLOSE_REQ  := TRUE;

               // set V2.1, V2.2
               // --------------
               "AM_SET_V2"(act_phase := "APC".SHUT_DOWN);

               // check end condition
               //--------------------
               IF NOT "LT".V1_OPEN THEN  // closed ? 
                   #end_of_step[0] := true;                            
               END_IF;

               #next_step[0] := 800; 


   //-step-800---level--0-------------------------------------------------------------                                                 
   //            SD: do leak test
   //---------------------------------------------------------------------------------                                                 
           800 :                                                  
               IF #next_step[0] = #active_step[0] THEN                       
                   "APC".TI[0] := 0;                              // start time for leak test                              
                   #prs_leak_test_start := "AV".ACT_PRS_FCH;           // save start pressure 
               END_IF;
               (*
               IF APC.TI[0] >= 3 THEN
                   DC.P1_ON := FALSE;
               END_IF;      
               *)
               #par_time := REAL_TO_INT ("PAR_MAIN".SD_LEAKTEST_TME);
               "APC".ACT_TME_STE := #par_time - "APC".TI[0];

               //store pressure value before leak test is starting (CDP)
               //-------------------------------------------------------
               "DIS".ACT_FNC_PRS_BEF_LKT :=  #prs_leak_test_start;

               // set V2.1, V2.2
               // --------------
               "AM_SET_V2"(act_phase := "APC".SHUT_DOWN);

               // leakrate = (p2-p1)*V/t
               // ----------------------
               IF ("APC".TI[0] > 0) THEN 
                   "AV".LRT_EKZ := ("AV".ACT_PRS_FCH - #prs_leak_test_start) * ("CNF".VOLUME_LEAK_TEST + "CNF".VOLUME_MAIN_FIL) / INT_TO_REAL("APC".TI[0]);
               END_IF;

               IF ("AV".LRT_EKZ < 0.0) THEN
                   "AV".LRT_EKZ := 0.0;
               END_IF;

               // show actual values
               // ------------------
               "DIS".ACT_LEAKR_FNC := "AV".LRT_EKZ;
               "APC".ACT_TME_STE   := #par_time - "APC".TI[0];


               IF ("APC".TI[0]>= #par_time) THEN                   // time for leak test ? 
                   #end_of_step[0] := true;                            
               END_IF;

               #next_step[0] := 900; 


   //-step-900---level--0-------------------------------------------------------------                                                 
   //            SD: check for max. leak rate
   //---------------------------------------------------------------------------------                                                 
           900 :                                                  
               IF ("AV".LRT_EKZ > "PAR_MAIN".SD_MAX_LEAKRATE) THEN  // max. leakrate ?
                   "FLT".PD_LEAKTEST := TRUE;
                   "APC".OP_MSG := "OP_MSG".SD_CHECK_LEAK_RATE;
                   #end_of_step[0] := true;                      // next step                            
               ELSE;
                   "APC".OP_MSG := "OP_MSG".BLANK;
                   #end_of_step[0] := true;                      // next step                            
               END_IF;

               #next_step[0] := 950;

   //-step-950---level--0-------------------------------------------------------------                                                 
   //            SD: check if gate valve is open
   //---------------------------------------------------------------------------------                                                 
           950 :                                                  
               IF NOT "LT".V7_OPEN THEN
                   IF NOT "FLT".PD_GATE_VALVE_CLOSED THEN 
                       "LT".AUTO_OP_CALL         := TRUE;    //set auto OP call once 
                   END_IF;
                   "FLT".PD_GATE_VALVE_CLOSED    := TRUE;
                   "APC".OP_MSG                  := "OP_MSG".OPEN_GATE_VALVE;  
               ELSE
                   "FLT".PD_GATE_VALVE_CLOSED    := FALSE;
                   "APC".OP_MSG                  := "OP_MSG".BLANK;   
                   #end_of_step[0]              := true;                      // next step                            

               END_IF;

               #next_step[0] := 1000;

   //-step-1000---level--0------------------------------------------------------------                                                 
   //            SD: wait until venting
   //---------------------------------------------------------------------------------                                                 
          1000 :                                                  
               IF #next_step[0] = #active_step[0] THEN                       
                   "APC".TI[0]       := 0;                                                           
                   "APC".OP_MSG      := "OP_MSG".SD_WAIT_TILL_VENTING;   
                   "LT".AUTO_OP_CALL := FALSE;        
               END_IF;

               //show remainig time of this step
               //-------------------------------
               "APC".ACT_TME_STE   := (REAL_TO_INT("PAR_MAIN".SD_WAIT_UNTIL_VENT)) - "APC".TI[0];

               //check end condition
               //-------------------
               IF ("APC".TI[0] >= (REAL_TO_INT("PAR_MAIN".SD_WAIT_UNTIL_VENT))) THEN
                   #end_of_step[0]  := true;                      // next step                            
               END_IF;

               #next_step[0] := 1100;

   //-step-1100---level--0------------------------------------------------------------                                                 
   //            SD: check if heater temperature is below pyrometer range
   //---------------------------------------------------------------------------------                                                 
          1100 :                                                  
               IF #next_step[0] = #active_step[0] THEN                       
                   "APC".OP_MSG  := "OP_MSG".SD_WAIT_UNTIL_COOL_DN;   
               END_IF;

               //check end condition
               //-------------------
               IF ("AV".ACT_HTR_1_TMP < "CNF".HTR_1_TMP_RANGE_LOW + 5.0) THEN
                   #end_of_step[0]  := true;                      // next step                            
               END_IF;

               #next_step[0] := 1200;

   //-step-1200--level--0-------------------------------------------------------------                                                 
   //            SD: vent furnace
   //---------------------------------------------------------------------------------                                                 
           1200 :                                                  
               IF #next_step[0] = #active_step[0] THEN                       
                   "APC".OP_MSG  := "OP_MSG".SD_VENTING;   
               END_IF;

               //stop pump only when no filter cleaning is triggered
               //---------------------------------------------------
               IF NOT "DV".FIL_FSH_REQ_AFTER_SD THEN
                   "DC".P1_ON := FALSE;                               // stop main pump
               END_IF;

               //vent furnace to atmospheric pressure
               //------------------------------------
               IF "DV".APS_GCH_DELAYED THEN
                   "DC".V4_OP    :=  FALSE;
               ELSE
                   "DC".V4_OP    :=  TRUE;
               END_IF;

               //check end condition
               //-------------------
               IF (NOT "DC".V4_OP AND NOT "PDO".V4) THEN
                   #end_of_step[0] := true;                          // next step                            
               END_IF;         

               #next_step[0] := 1300;

   //-step-1300---level--0------------------------------------------------------------                                                 
   //            SD: wait after venting
   //---------------------------------------------------------------------------------                                                 
          1300 :                                                  
               IF #next_step[0] = #active_step[0] THEN                       
                   "APC".TI[0]   := 0;                                                           
                   "APC".OP_MSG  := "OP_MSG".SD_WAIT_AFT_VENT;   
               END_IF;

               //show remainig time of this step
               //-------------------------------
               "APC".ACT_TME_STE   := (REAL_TO_INT("PAR_MAIN".SD_WAIT_AFT_VENT)) - "APC".TI[0];

               //check end condition
               //-------------------
               IF ("APC".TI[0] >= (REAL_TO_INT("PAR_MAIN".SD_WAIT_AFT_VENT))) THEN
                   #end_of_step[0]  := true;                      // next step                            
               END_IF;

               #next_step[0] := 1400;

   //-step-1400--level--0-------------------------------------------------------------                                                 
   //            SD: start idle mode
   //---------------------------------------------------------------------------------                                                 
           1400 :

               "APC".OP_MSG      := "OP_MSG".BLANK;
               "APC".ACT_TME_STE := 0;
               "FLT".PD_LEAKTEST := FALSE;

               "DC".MOD_ID := TRUE;                               // switch to idle 

               #next_step[0] := 1400;                            // E N D

   //-error------level--0---------------------------------------------------(error in level 0)-------------
       ELSE:                                                        
           //error code                                                //do error code
           ;        
   //------------------------------------------------------------------------------------------------------
       END_CASE;


       #start_previous := #start;                                    //save start input for next call 
       #cont_previous := "APC".CONT;                                  //save cont input for next call 
       #resume_previous := "APC".RESUME;                              //save resume input for next call
       #jump_previous := "APC".JUMP;                                  //save jump input for next call
       #single_previous := "APC".SINGLE;                              //save single input for next call
END_FUNCTION_BLOCK

FUNCTION_BLOCK "AM_RE"   // FB204, SCL
{ S7_Optimized_Access := 'FALSE' }
VERSION : 0.0
// --------------------------------------------------------------------------------
//     program     :    AM_RE
//     description :    apc removal module  
//     name        :    L. Vogel
//     date        :    27.06.2012
// 
//     revision    : 
//     name        :   
//     date        :    
// 
//                     (c)PVA TePla AG
//     --------------------------------------------------------------------------------
   VAR_INPUT
      start : Bool;   // start sequence, activate step 10 (impulse triggered)
   END_VAR
   VAR
      start_previous : Bool;   // start input value of last call
      cont_previous : Bool;   // cont input value of last call
      resume_previous : Bool;   // resume input value of last call
      jump_previous : Bool;   // jump input value of last call
      single_previous : Bool;   // single input value of last call
      active_step : Array[0..7] of Int;   // active step number for sequence level 0..7
      next_step : Array[0..7] of Int;   // next step number for sequence level 0..7
      hold_step : Array[0..7] of Int;   // step number of step on hold
      end_of_step : Array[0..7] of Bool;   // active step is done flag for sequence 0..7
      EndOfStep : Bool;   // default value for active step is done flag
      cont_enable : Array[0..7] of Bool;   // enable continue function
      ContEnable : Bool;   // default value for enable continue function
      xt_removed : Bool;
      cr_lft_man_off : Bool;
      prg_cyc_cnt : Int;
      xt_start_pos : Real;   // crystal position at start of removal
      cr_start_rot : Real;   // crucible rotation at start of removal
      cr_start_pos : Real;   // crucible position at start of removal
      htr_start_temp : Real;   // heater temperature at start of removal
      set_body_length : Real;   // set point of body length
   END_VAR
BEGIN


       "APC".STATUS := "APC".REMOVAL;                                  // set apc status               

       "AM_SEQUENCE_CTL" (start_p            := #start,               // control sequence
                        start_previous_p   := #start_previous,
                        cont_previous_p    := #cont_previous, 
                        resume_previous_p  := #resume_previous,
                        jump_previous_p    := #jump_previous,
                        single_previous_p  := #single_previous,
                        active_step_p      := #active_step, 
                        next_step_p        := #next_step,
                        hold_step_p        := #hold_step, 
                        end_of_step_p      := #end_of_step, 
                        cont_enable_p      := #cont_enable); 

       //set point magnet
       //----------------
       "AC".SET_MAG_1_CUR    :=  "AV".SET_MAG_1_CUR;
       "AC".SET_MAG_2_CUR    :=  "AV".SET_MAG_2_CUR;  
       "DC".MAG_ON           := ("AC".SET_MAG_1_CUR > 0.0);

       //Set the "Oxidation valve" in all Phases
       "DC".V21_OP:= DINT_TO_BOOL(REAL_TO_DINT("PAR_MAIN".RC_V21_OPEN));

       CASE #active_step[0] OF    //sequence level_0
   //step--0-----level--0-------------------------------------------------off--(sequence off)--------------
           0    :                                                  
                #next_step[0] := 0;

   //step--1-----level--0-------------------------------------------------hold-(test sequence)-------------
           1   :                                                       
               IF #next_step[0] = #active_step[0] THEN                   //init step     
                   //init code
                   ; 
               END_IF;

               //step code                                             //do step
               ;

   //-step-10----level--0----------------------------------------------main-(start sequence)---------------                                                 

   //-step-10----level--0-------------------------------------------------------------                                                 
   //            RE: init removal sequence
   //---------------------------------------------------------------------------------                                                 
           10  :

               // save data of grown body (for 2nd body)
               // --------------------------------------
               IF ("APC".RE_WHILE_BY = TRUE) THEN    // removal started during body ?
                   "APC".RE_WHILE_BY := FALSE;
                   "APC".LEN2_CALC   := FALSE;
                   "APC".PNBDY       := TRUE;
                   "APC".SUTDN       := TRUE;
                   "CM_SAVE_GROWN_BY" (with_endcone := FALSE,
                                     dia          := "AC".SET_XT_DIA,
                                     len          := "AV".ACT_XT_LEN);

               END_IF;

               // init vacuum system
               // ------------------
               "DC".V3_OP    := FALSE;
               "DC".V4_OP    := FALSE;
               "DC".V5_OP    := TRUE;
               "DC".V6_OP    := FALSE;
               "DC".V8_OP    := FALSE;
               "DC".V11_OP   := FALSE;
               "DC".V11_CL   := TRUE;
               "DC".V12_OP   := FALSE;
               "DC".V13_OP   := FALSE;
               "DC".V20_OP   := FALSE;
               "DC".V22_OP   := FALSE;
               "DC".V24_OP   := FALSE;
               "DC".P1_ON    := TRUE;                        // start main pump
               "DC".P3_ON    := FALSE;
               "DC".V3_4_OP  := FALSE;
               "DC".V1_1_REL := FALSE;

               "DC".V3_2_OP  := FALSE;                       // vacuum valve feeder
               #prg_cyc_cnt := 0;

               // init drives
               // -----------
               "DC".XT_LFT_UP    := TRUE;                                    // crystal lift up
               "DC".XT_LFT_DN    := FALSE;
               "DC".XT_LFT_FST   := FALSE;
               "DC".XT_ROT_CW    := "BM_ROT_DRV_DIR_DB".ROT_DIR;               //1 = cw
               "DC".XT_ROT_CCW   := NOT "BM_ROT_DRV_DIR_DB".ROT_DIR;           //0 = ccw

               "DC".CR_LFT_UP    := FALSE;                                   // stop crucible lift
               "DC".CR_LFT_DN    := FALSE;
               "DC".CR_LFT_FST   := FALSE;
               "DC".CR_ROT_CW    := NOT "BM_ROT_DRV_DIR_DB".ROT_DIR;           //0 = cw
               "DC".CR_ROT_CCW   := "BM_ROT_DRV_DIR_DB".ROT_DIR;               //1 = ccw

               "AC".SET_XT_SPD   := "KYA".SET_XT_SPD;                
               "AC".SET_XT_ROT   := "KYA".SET_XT_ROT;
               "AC".SET_CR_SPD   := 0.0;
               "AC".SET_CR_ROT   := "KYA".SET_CR_ROT;

               // init heater
               // -----------
               "DC".HTR_1_ON     := TRUE;                                    // heater off
               "DC".HTR_2_ON     := TRUE;
               "DC".HTR_3_ON     := FALSE;

               // AC.SET_HTR_1_PWR := 0.0;                 do not set, loop is on
               // AC.SET_HTR_2_PWR := 0.0;
               // AC.SET_HTR_3_PWR := 0.0;

               //mobile feeder
               //-------------
               "DC".MOB_FDR_MVE_IN_SEQ_ON    :=  FALSE;
               IF ("LT".MOB_FDR_DCK_DONE AND ("DV".FDG_MVE_IN_SEQ_DONE OR NOT "DV".FDG_MVE_OUT_SEQ_DONE)) THEN 
                   "DC".MOB_FDR_MVE_OUT_SEQ_ON   :=  TRUE;
               ELSE
                   "DC".MOB_FDR_MVE_OUT_SEQ_ON   :=  FALSE;
               END_IF;
               "DC".MOB_FDR_VIB_ON           :=  FALSE;
               "FLT".MOB_FDR_NOT_DCK         :=  FALSE;
               "FLT".MOB_FDR_STP_PARA        :=  FALSE;

               // init magnet
               // -----------
               "DC".MAG_ON               := ("AC".SET_MAG_1_CUR > 0.0);       
               "AC".SET_MAG_1_CUR        :=  "KYA".SET_MAG_1_CUR;
               "AC".SET_MAG_2_CUR        :=  "KYA".SET_MAG_2_CUR;

               // init control loops
               // ------------------
               "DC".CTL_DIA_ON           := FALSE;       // all control loops off
               "DC".CTL_GRW_RTE_ON       := FALSE;
               "DC".CTL_PULL_RTE_ON      := FALSE;
               "DC".CTL_CRUC_ROT_ON      := FALSE;
               "DC".CTL_MLT_LVL_ON       := FALSE;
               "DC".CTL_MLT_1_TMP_ON     := FALSE;
               "DC".CTL_MLT_2_TMP_ON     := FALSE;
               "DC".CTL_MLT_DRIFT_ON     := FALSE;
               "DC".CTL_GAP_ON           := FALSE;

               "DC".CTL_HTR_1_TMP_ON     := TRUE;        // heater temp. loop on
             //DC.CTL_HTR_2_TMP_ON     := FALSE;

               "DC".SET_HTR_1_TMP_ABS    := TRUE;        // disable inc functions
               "DC".SET_HTR_2_PWR_ABS    := TRUE;

               "DC".CTL_PRS_ON           := TRUE;        // pressure loop on 

               "DC".CTL_SI_FDR_ON        := FALSE;
               "DC".CTL_DOP_FDR_ON       := FALSE;

               "AC".SET_XT_DIA           := 0.0;
               "AC".SET_GRW_RTE          := 0.0;
               "AC".SET_AVG_SPD          := 0.0;
               "AC".SET_AVG_CRUC_ROT     := 0.0;
               "AC".SET_MLT_LVL_LSR      := 0.0;
               "AC".SET_MLT_1_TMP        := 0.0;
               "AC".SET_MLT_2_TMP        := 0.0;
               "AC".SET_HTR_1_TMP_INC    := 0.0;
               "AC".SET_HTR_2_PWR_INC    := 0.0;
               "AC".SET_HTR_1_TMP        := "DIS".ACT_HTR_1_TMP;   //presetting of AC set point variable

               // init measurement system
               // -----------------------
               "DC".CAM_ISP_ON           := FALSE;       //inspection off
               "DC".CAM_INIT             := FALSE;
             //DC.CAM_MLT              := FALSE;
             //DC.CAM_DIP              := FALSE;
             //DC.CAM_DIA              := TRUE;
               "DC".CAM_SEL_1            := TRUE;
               "DC".CAM_SEL_2            := FALSE;

               "DC".LSR_ON               := FALSE;       // laser off
               "DC".MCC_ON               := FALSE;       // melt contact control off
               "DC".MCC_TST_ON           := FALSE;

               // init Si feeder system
               // ---------------------
               "DC".SI_FDR_ON            := FALSE;       // feeder off
               "DC".DOP_FDR_ON           := FALSE;

               "AC".SET_FDR_SI           := 0.0;
               "AC".SET_FDR_DOP          := 0.0;

               "LT".SHOW_HTR_1_TRG_TMP   := FALSE;

               // init lamp on control cabinet
               // ----------------------------
               "DV".LMP_OR               := FALSE;

               // enable automatic mode
               // ---------------------
               "DC".MOD_AUT_ENB          := TRUE;    

               #end_of_step[0]          := true;                            
               #next_step[0]            := 100;

   //-step-100---level--0-------------------------------------------------------------                                                 
   //            RE: wait for automatic mode
   //---------------------------------------------------------------------------------                                                 
           100 :                                                     
               IF #next_step[0] = #active_step[0] THEN
                   "APC".OP_MSG := "OP_MSG".WAIT_FOR_AUTO;                                                  
               END_IF;

               IF "APC".AUTOMATIC THEN                   // automatic mode ?
                   #end_of_step[0] := true;                            
               // calculate actual length
               // -----------------------
               ELSIF "PDI".MCC_CONTACT_XT THEN 
                   IF ("APC".BYRST) THEN
                       #set_body_length := "AV".SET_XT_LEN_BDY2;        // 2nd body
                   ELSE
                       #set_body_length := "PAR_MAIN".BY_XT_LEN;
                   END_IF;
                   "AM_CALC_LENGTH" (start_pos       := "AV".XT_POS_AT_START_BY,
                                   actual_pos      := "AV".ACT_XT_POS,
                                   total_len       := #set_body_length,
                                   actual_len      => "AV".ACT_XT_LEN,
                                   actual_len_prc  => "AV".ACT_XT_LEN_PRC);
               END_IF;

               #next_step[0] := 200;

   //-step-200---level--0-------------------------------------------------------------                                                 
   //            RE: start time
   //---------------------------------------------------------------------------------                                                 
           200 :                                                     
               "APC".ACT_TME_PROC    := 0;               // start process time
               "APC".ACT_TME_STE     := 0;               // reset time of step
               "APC".TI[0]           := 0;               // start waiting time
               "APC".OP_MSG          := "OP_MSG".BLANK;                                                  

               #end_of_step[0]  := true;                            

               #next_step[0]    := 300;

   //-step-300---level--0-------------------------------------------------------------                                                 
   //            RE: raise heater 1 temperature set point and lower crucible rotation
   //---------------------------------------------------------------------------------                                                 
           300 :                                                     
               IF #next_step[0] = #active_step[0] THEN  
                   "APC".TI[0]       := 0;        
                   "APC".OP_MSG      := "OP_MSG".RE_HTR_TMP_RSD;             
                   //reset initial temperature and power setpoints
                   //---------------------------------------------
                   "DIS".HTR_1_TMP_SET_PHA_STR   :=  0.0;
                   "DIS".HTR_2_PWR_SET_PHA_STR   :=  0.0;
                   "AC".SET_HTR_1_TMP            :=  "DIS".ACT_HTR_1_TMP;
                   #cr_start_rot                :=  "AC".SET_CR_ROT;
                   #htr_start_temp              :=  "AC".SET_HTR_1_TMP;
               END_IF;

               // calculate all setpoints for this step
               // -------------------------------------                                      
               "AM_PAR_FNC_RE"();

               //switch melt contact control on
               //------------------------------
               "DC".MCC_ON := TRUE;                       

               // calculate actual length
               // -----------------------
               IF "PDI".MCC_CONTACT_XT THEN 
                   IF ("APC".BYRST) THEN
                       #set_body_length := "AV".SET_XT_LEN_BDY2;        // 2nd body
                   ELSE
                       #set_body_length := "PAR_MAIN".BY_XT_LEN;
                   END_IF;
                   "AM_CALC_LENGTH" (start_pos       := "AV".XT_POS_AT_START_BY,
                                   actual_pos      := "AV".ACT_XT_POS,
                                   total_len       := #set_body_length,
                                   actual_len      => "AV".ACT_XT_LEN,
                                   actual_len_prc  => "AV".ACT_XT_LEN_PRC);
               END_IF;

               //write target heater 1 temperature set point
               //-------------------------------------------
               "DIS".RE_HTR_1_TRG_SET_TMP    :=  "AV".SET_DIP_TMP + 10.0;
               "LT".SHOW_HTR_1_TRG_TMP       :=  TRUE;

               //heater 1 temperature set point ramp
               //-----------------------------------
               IF ("SysTick1s" AND ("DIS".RE_HTR_1_TRG_SET_TMP > "AC".SET_HTR_1_TMP)) THEN
                   "AC".SET_HTR_1_TMP := "AC".SET_HTR_1_TMP + ("CNF".RE_RMP_RTE_HTR / 60.0);
               END_IF;

               //crucible rotation set point ramp
               //--------------------------------
               IF ("SysTick1s" AND ("AC".SET_CR_ROT > "PAR_MAIN".RC_CR_ROT)) THEN 
                   "AC".SET_CR_ROT := "AC".SET_CR_ROT - ("CNF".RE_RMP_RTE_CR_ROT / 60.0);
               END_IF;

               //switch to next step when when actual temp is 20K above start temp
               //-----------------------------------------------------------------
               IF ("AV".ACT_HTR_1_TMP >= (#htr_start_temp + 20.0)) THEN    
                   #end_of_step[0] := true;                            
               END_IF;

               #next_step[0] := 400; 

   //-step-400---level--0-------------------------------------------------------------                                                 
   //            RE: crucible lift down
   //---------------------------------------------------------------------------------                                                 
           400 :                                                     
               IF #next_step[0] = #active_step[0] THEN                       
                   "APC".TI[0]       := 0;           
                   "APC".TI[1]       := 0;          
                   "APC".OP_MSG      := "OP_MSG".RE_CR_LWD;
                   #cr_start_pos    := "AV".ACT_CR_POS;
                END_IF;

               // calculate all setpoints for this step
               // -------------------------------------                                      
               "AM_PAR_FNC_RE"();

               // calculate actual length
               // -----------------------
               IF "PDI".MCC_CONTACT_XT THEN 
                   IF ("APC".BYRST) THEN
                       #set_body_length := "AV".SET_XT_LEN_BDY2;        // 2nd body
                   ELSE
                       #set_body_length := "PAR_MAIN".BY_XT_LEN;
                   END_IF;
                   "AM_CALC_LENGTH" (start_pos       := "AV".XT_POS_AT_START_BY,
                                   actual_pos      := "AV".ACT_XT_POS,
                                   total_len       := #set_body_length,
                                   actual_len      => "AV".ACT_XT_LEN,
                                   actual_len_prc  => "AV".ACT_XT_LEN_PRC);
               END_IF;

               //heater 1 temperature set point ramp
               //-----------------------------------
               IF ("SysTick1s" AND ("DIS".RE_HTR_1_TRG_SET_TMP > "AC".SET_HTR_1_TMP)) THEN
                   "AC".SET_HTR_1_TMP := "AC".SET_HTR_1_TMP + ("CNF".RE_RMP_RTE_HTR / 60.0);
               END_IF;

               //crucible rotation set point ramp
               //--------------------------------
               IF ("SysTick1s" AND ("AC".SET_CR_ROT > "PAR_MAIN".RC_CR_ROT)) THEN 
                   "AC".SET_CR_ROT := "AC".SET_CR_ROT - ("CNF".RE_RMP_RTE_CR_ROT / 60.0);
               END_IF;

               //crucible lift down
               //------------------
               "DC".CR_LFT_DN    :=  TRUE;
               "AC".SET_CR_SPD   :=  "CNF".RE_CR_SPD;

               //check end condition
               //-------------------
               IF ("APC".TI[0] > 120) THEN                                       //min. time of this step is 120sec.
                   IF (NOT "PDI".MCC_CONTACT_XT OR ("APC".TI[0] > 600)) THEN       //melt contact lost or max. time of this step over
                       IF ("APC".TI[1] > 5)  THEN                                //delay end of step 5 sec. after melt contact lost
                           #end_of_step[0] := true;                            
                       END_IF;
                   ELSE
                       "APC".TI[1] := 0;
                   END_IF;
               END_IF;

               #next_step[0] := 500; 

   //-step-500---level--0-------------------------------------------------------------                                                 
   //            RE: crystal is out of melt - move up with low speed
   //---------------------------------------------------------------------------------                                                 
           500 :                                                     
               IF #next_step[0] = #active_step[0] THEN                       
                   "APC".TI[0]       :=  0;                     
                   #xt_start_pos    :=  "AV".ACT_XT_POS; 
                   "APC".OP_MSG      :=  "OP_MSG".RE_CRYSTAL_UP;
                END_IF;

               //calculate all setpoints for this step
               //-------------------------------------                                      
               "AM_PAR_FNC_RE"();

               //heater 1 temperature set point ramp
               //-----------------------------------
               IF ("SysTick1s" AND ("DIS".RE_HTR_1_TRG_SET_TMP > "AC".SET_HTR_1_TMP)) THEN
                   "AC".SET_HTR_1_TMP := "AC".SET_HTR_1_TMP + ("CNF".RE_RMP_RTE_HTR / 60.0);
               END_IF;

               //crucible rotation set point ramp
               //--------------------------------
               IF ("SysTick1s" AND ("AC".SET_CR_ROT > "PAR_MAIN".RC_CR_ROT)) THEN 
                   "AC".SET_CR_ROT := "AC".SET_CR_ROT - ("CNF".RE_RMP_RTE_CR_ROT / 60.0);
               END_IF;

               //crystal lift up with selectable low speed
               //-----------------------------------------
               "AC".SET_XT_SPD := "PAR_MAIN".RC_XT_LFT_SPD;

               //stop crucible lift
               //------------------
               "DC".CR_LFT_DN    :=  FALSE;
               "AC".SET_CR_SPD   :=  0.0;

               //check end condition
               //-------------------
               #next_step[0] := 600; 

               // time till end of this step
               // --------------------------
               "APC".ACT_TME_STE := (REAL_TO_INT("PAR_MAIN".RC_XT_LFT_TME) * 60) - "APC".TI[0];

               //raise time with low speed is over
               //---------------------------------
               IF ("APC".TI[0] > (REAL_TO_INT("PAR_MAIN".RC_XT_LFT_TME) * 60)) THEN        
                   #end_of_step[0]  := true;       

               //final position above melt is already reached
               //--------------------------------------------
               ELSIF (("AV".ACT_XT_POS < (#xt_start_pos - "PAR_MAIN".RC_XT_POS)) OR ("AV".ACT_XT_POS < ("PAR_MAIN".MCONST_LIM_XTAL_UP + 10.0))) THEN        
                   #end_of_step[0]  := true; 
                   #next_step[0]    := 700; 
               END_IF;

   //-step-600---level--0-------------------------------------------------------------                                                 
   //            RE: crystal to final position
   //---------------------------------------------------------------------------------                                                 
           600 :                                                     
               IF #next_step[0] = #active_step[0] THEN                       
                   "APC".OP_MSG  := "OP_MSG".RE_CRYSTAL_TO_POS;
                   "DC".MCC_ON   := FALSE;                       // melt contact control off
               END_IF;

               // calculate all setpoints for this step
               // -------------------------------------                                      
               "AM_PAR_FNC_RE"();

               //raise crystal with faster speed in gate chamber
               //-----------------------------------------------   
               "DC".XT_LFT_FST   := TRUE;
               "AC".SET_XT_SPD   := "CNF".RE_XT_SPD_FST;

               //check end condition
               //-------------------
               IF (("AV".ACT_XT_POS < (#xt_start_pos - "PAR_MAIN".RC_XT_POS)) OR ("AV".ACT_XT_POS < ("PAR_MAIN".MCONST_LIM_XTAL_UP + 10.0))) THEN
                   #end_of_step[0] := true;                            
               END_IF;

               #next_step[0] := 700; 

   //-step-700---level--0-------------------------------------------------------------                                                 
   //            RE: crystal in gate chamber - close gate valve
   //---------------------------------------------------------------------------------                                                 
           700 :                                                     
               IF #next_step[0] = #active_step[0] THEN                       
                   "APC".OP_MSG          := "OP_MSG".CLOSE_GATE_VALVE;
                   "LT".AUTO_OP_CALL     := TRUE;
                   "DC".MCC_ON           := FALSE;                       // melt contact control off
               END_IF;

               // calculate all setpoints for this step
               // -------------------------------------                                      
               "AM_PAR_FNC_RE"();

               //stop crystal lift
               //----------------
               "DC".XT_LFT_UP  := FALSE;                     
               "DC".XT_LFT_FST := FALSE;
               "AC".SET_XT_SPD := 0.0;                

               //check end_condition
               //-------------------
               IF ("LT".V7_CLOSE AND NOT "LT".V7_OPEN AND "DV".LS_V7_DN_DLY) THEN         // V7 closed ?
                   "DC".V5_OP            := FALSE;               //close valve V5
                   "DC".V6_OP            := TRUE;                //open valve V6
                   #end_of_step[0]      := true;                            
               END_IF;

               #next_step[0] := 800; 

